(* IEC 61131-3 sources: CodesysTest/alpha/export/ObjectHandling/FB_CollectionHandlerOEEQualityFaults.pou, 4 files *)

(* ---- FB_CollectionHandlerOEEQualityFaults.pou.st ---- *)
(*#-#-#-#-#-#-#-#-#-#---Declaration---#-#-#-#-#-#-#-#-#-#-#-#-#*)

FUNCTION_BLOCK FB_CollectionHandlerOEEQualityFaults
VAR_INPUT
END_VAR
VAR_OUTPUT
	totalObj : INT;
	faultExempt : BOOL;
	collection : ARRAY[0..GlobalObjects.MAX_FAULTS] OF IFault;
END_VAR
VAR
	_objNames : ARRAY[0..GlobalObjects.MAX_FAULTS] OF STRING;
END_VAR(*#-#-#-#-#-#-#-#-#-#---Implementation---#-#-#-#-#-#-#-#-#-#-#-#-#*)

//
//  FB_CollectionHandlerPassiveFaults
//  FB/Object Handling/FB_CollectionHandlerOEEExemptFaults
//
//  Created by Ben Hess on 05/31/2022.
//  Copyright (C) 2021 Sharp Packaging Systems By Pregis. All rights reserved.
//

(* ---- AckAll.m.st ---- *)
(*#-#-#-#-#-#-#-#-#-#---Declaration---#-#-#-#-#-#-#-#-#-#-#-#-#*)

METHOD AckAll
VAR_INPUT
END_VAR
VAR
	_cast : IFault;
	_fault : IFault;
	_j : INT;
END_VAR(*#-#-#-#-#-#-#-#-#-#---Implementation---#-#-#-#-#-#-#-#-#-#-#-#-#*)

// For each active fault in the array, ack it.
FOR _j:= 0 TO totalObj - 1 DO
	IF (__QUERYINTERFACE(collection[_j], _cast)) THEN
		_cast.Ack();
	ELSE
		RETURN;
	END_IF
END_FOR

(* ---- AddObject.m.st ---- *)
(*#-#-#-#-#-#-#-#-#-#---Declaration---#-#-#-#-#-#-#-#-#-#-#-#-#*)

METHOD AddObject
VAR_INPUT
	obj : IFault;
END_VAR
VAR
	_j : INT;
END_VAR(*#-#-#-#-#-#-#-#-#-#---Implementation---#-#-#-#-#-#-#-#-#-#-#-#-#*)

// Add the active fault to the array
FOR _j := 0 TO totalObj DO
	IF collection[_j] = Obj THEN
		// object pointer matches - it's already in here
		RETURN;
	END_IF
END_FOR

IF totalObj < GlobalObjects.MAX_FAULTS THEN
	collection[totalObj]:= Obj;
	_objNames[totalObj]:= Obj.InstanceName;
	totalObj:= totalObj + 1;
END_IF
faultExempt := TRUE;

(* ---- RemoveObject.m.st ---- *)
(*#-#-#-#-#-#-#-#-#-#---Declaration---#-#-#-#-#-#-#-#-#-#-#-#-#*)

METHOD RemoveObject
VAR_INPUT
	obj : IFault;
END_VAR
VAR
	_i : INT;
	_j : INT;
END_VAR
(*#-#-#-#-#-#-#-#-#-#---Implementation---#-#-#-#-#-#-#-#-#-#-#-#-#*)

FOR _i:= 0 TO totalObj DO
	IF collection[_i] = obj THEN
		// object pointer matches - get rid of it
		FOR _j := _i TO totalObj DO
			collection[_J] := collection[_j+1];
			_objNames[_J]:= _objNames[_j+1];
		END_FOR
		totalObj := totalObj - 1;
		IF totalObj = 0 THEN
			faultExempt := FALSE;
		END_IF
		RETURN;
	END_IF
END_FOR
